ADAPTER ASupply (* Adapter Interface *)
  (* Standard: 61499-1 *)
  (* Version 1.0, 2018-07-17, az *)
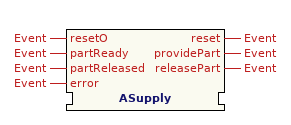
  EVENT_INPUT
    resetO; (* Request from Socket *)
    partReady; (* Response from Socket *)
    partReleased;
    error;
  END_EVENT
  EVENT_OUTPUT
    reset; (* Confirmation from Plug *)
    providePart; (* Indication from Plug *)
    releasePart;
  END_EVENT
  SERVICE SOCKET/PLUG (* Adapter Interface *)
    SEQUENCE request_confirm
      SOCKET.REQ(REQD) -> PLUG.REQ(REQD);
      PLUG.CNF(CNFD) -> SOCKET.CNF(CNFD);
    END_SEQUENCE
    SEQUENCE indication_response
      PLUG.IND(INDD) -> SOCKET.IND(INDD);
      SOCKET.RSP(RSPD) -> PLUG.RSP(RSPD);
    END_SEQUENCE
  END_SERVICE
END_ADAPTER
